{attribute 'qualified_only'}
VAR_GLOBAL
END_VAR

(* stored: Version 1.1.0.1, ProductVersion 3.1.4024.14
   GVL GVL: Id {1d76f2ad-27fd-464a-b815-9cfe8ba938f8} *)
